VANND_L22_V0342 722.11 BOOL
VANND_L22_V0405 722.09 BOOL
VANND_L22_V0505 722.10 BOOL
VASK_SLANGE 723.12 BOOL  ; SLANGE OENSKES VASKET IC79
VASK_SLANGE_COM_BIT 1150.02 BOOL  ; SLANGE SKAL INNGAA I C79
VENTILFEIL_SIRK_K1 1309.04 BOOL
VENTILFEIL_SIRK_K2 1319.04 BOOL
VENTILFEIL_SIRK_K3 1329.04 BOOL
VS80_K1_HJ_RAP_2STA 901.07 BOOL
VS80_K2_HJ_RAP_2STA 911.07 BOOL
VS80_K3_HJ_RAP_2STA 921.07 BOOL
VST60_K1_KL_INN_N6 2841.08 BOOL
VST60_K1_TR5_N6 2865.02 BOOL
VST60_K2_KL_AVSL 1816.09 BOOL
VST60_K2_KL_INN 1816.08 BOOL
VST80K1_BET_FLOWKONTROLL 1309.07 BOOL  ; BETINGELER START TID FOR FLOWKONTROLL INN
VST80K1_ER_VENT_FLOW D8631 UINT  ; ER- VERDI VENTETID FOER FLOWKONTROLL STARTER
VST80K1_FLOWFEIL 1309.09 BOOL  ; FOR LAV FLOW I RETUR
VST80K1_FLOWKONTROLL 1309.08 BOOL
VST80K1_FLOWKONTROLL_S T0933 BOOL  ; TID MED FOR LAV FLOW I RETUR FOER ALARM SLAAR INN
VST80K1_MAX_DIF_FLOWKONTROLL D8616 UINT  ; MAXIMAL DIFFERANSE MELLOM TUR OG RETURFLOW
VST80K1_PRS_VENT_FLOW D8630 UINT  ; PRS VENTETID FOER FLOWKONTROLL STARTER
VST80K2_BET_FLOWKONTROLL 1319.07 BOOL  ; BETINGELER START TID FOR FLOWKONTROLL INN
VST80K2_ER_VENT_FLOW D8731 UINT  ; ER- VERDI VENTETID FOER FLOWKONTROLL STARTER
VST80K2_FLOWFEIL 1319.09 BOOL  ; FOR LAV FLOW I RETUR
VST80K2_FLOWKONTROLL 1319.08 BOOL
VST80K2_FLOWKONTROLL_S T0934 BOOL  ; TID MED FOR LAV FLOW I RETUR FOER ALARM SLAAR INN
VST80K2_MAX_DIF_FLOWKONTROLL D8716 UINT  ; MAXIMAL DIFFERANSE MELLOM TUR OG RETURFLOW
VST80K2_PRS_VENT_FLOW D8730 UINT  ; PRS VENTETID FOER FLOWKONTROLL STARTER
VST80K3_BET_FLOWKONTROLL 1329.07 BOOL  ; BETINGELER START TID FOR FLOWKONTROLL INN
VST80K3_ER_VENT_FLOW D8801 UINT  ; ER- VERDI VENTETID FOER FLOWKONTROLL STARTER
VST80K3_FLOWFEIL 1329.09 BOOL  ; FOR LAV FLOW I RETUR
VST80K3_FLOWKONTROLL 1329.08 BOOL
VST80K3_FLOWKONTROLL_S T0935 BOOL  ; TID MED FOR LAV FLOW I RETUR FOER ALARM SLAAR INN
VST80K3_MAX_DIF_FLOWKONTROLL D8816 UINT  ; MAXIMAL DIFFERANSE MELLOM TUR OG RETURFLOW
VST80K3_PRS_VENT_FLOW D8800 UINT  ; PRS VENTETID FOER FLOWKONTROLL STARTER
VST80_BIL1_VASKET 701.02 BOOL  ; BENYTTES TIL FLASH PAA VEGG VED BIL 1
VST80_BIL1_VASKET_TID_S T0114 BOOL  ; BENYTTES TIL AA RESET 701.02
VST80_BIL1_VASKET_TID_T 0114 NUMBER  ; BENYTTES TIL AA RESET 701.02
VST80_BIL21_VASKET_TID_S T0116 BOOL  ; BENYTTES TIL AA RESET 705.02
VST80_BIL2_VASKET 705.02 BOOL  ; BENYTTES TIL FLASH PAA VEGG VED BIL 2
VST80_BIL2_VASKET_TID_T 0116 NUMBER  ; BENYTTES TIL AA RESET 705.02
VST80_HENGER1_VASKET 703.02 BOOL  ; BENYTTES TIL FLASH PAA VEGG VED HENGER 1
VST80_HENGER1_VASKET_T 0115 NUMBER  ; BENYTTES TIL AA RESET 703.02
VST80_HENGER1_VASKET_TID_S T0115 BOOL  ; BENYTTES TIL AA RESET 703.02
VST80_HENGER2_VASKET 707.02 BOOL  ; BENYTTES TIL FLASH PAA VEGG VED HENGER 2
VST80_HENGER2_VASKET_T 0117 NUMBER  ; BENYTTES TIL AA RESET 707.02
VST80_HENGER2_VASKET_TID_S T0117 BOOL  ; BENYTTES TIL AA RESET 707.02
VST80_K1R_DIF_S 1308.02 BOOL  ; MENGEDIFFERANSE TUR RETUR FOR STOR
VST80_K1_0_STATUS 500.01 BOOL  ; XX
VST80_K1_0_ST_HJ1 400.00 BOOL
VST80_K1_0_ST_HJ2 400.01 BOOL
VST80_K1_0_ST_HJ3 400.02 BOOL
VST80_K1_1_STATUS 500.02 BOOL  ; Z
VST80_K1_1_ST_HJ1 400.03 BOOL
VST80_K1_1_ST_HJ2 400.04 BOOL  ; Z
VST80_K1_1_ST_HJ3 400.05 BOOL  ; Z
VST80_K1_1_ST_HJ4 400.06 BOOL  ; Z
VST80_K1_1_ST_HJ5 400.07 BOOL  ; Z
VST80_K1_1_ST_HJ6 400.08 BOOL  ; Z
VST80_K1_2_STAT 500.03 BOOL  ; Z
VST80_K1_2_ST_HJ1 400.09 BOOL  ; Z
VST80_K1_2_ST_HJ2 400.10 BOOL  ; Z
VST80_K1_AUT_NOEDSTOPP 1305.04 BOOL  ; NOEDSTOPPSIGNAL FRA VASKESTASJON KURS1
VST80_K1_AVLESE_FLOW D7990 INT
VST80_K1_AVLES_FLOW D8690 INT
VST80_K1_B8011_ER_CT D8040 CHANNEL  ; B8011 -VST80-KURS1. ER-VERDI KONDUKTIVITET I RETUR TIL VST
VST80_K1_B8012_ER_TT D8006 CHANNEL  ; B8012 -VST80-KURS1. ER-VERDI TEMPERATUR I RETUR TIL VST
VST80_K1_B8012_ER_TTR D8604 INT
VST80_K1_B8014_ER_TT D8000 CHANNEL  ; B8014 -VST80-KURS1. ER-VERDI TEMPERATUR I TUR TIL VST
VST80_K1_DIF_HYSTVERDI_OVERSKREDET 1308.01 BOOL  ; BENYTTES TIL AA SKAPE HYSTERESE VED FOR STOR MENDEFORSK. MELLOM TUR OG RETUR  1308.01=0=MENDEDIF OK
VST80_K1_DRIFT 500.00 BOOL  ; XX
VST80_K1_ER_COND D8600 CHANNEL  ; SKAL_RETTES_TIL_K1_KOND_ERVERDI
VST80_K1_FEIL 500.04 BOOL  ; Z
VST80_K1_FEILTID 500.05 BOOL  ; Z
VST80_K1_FORSINK_MENGDEDIF T0151 BOOL  ; TID SOM FORSINKER MENGDEDIF. STOPP AV FASE
VST80_K1_GRM_KONTR_VENT T0884 BOOL  ; VENT MED GRENSEMELKOVERVAAKING
VST80_K1_HJ10 902.01 BOOL
VST80_K1_HJ11 902.02 BOOL
VST80_K1_HJ12 902.03 BOOL
VST80_K1_HJ13 902.04 BOOL
VST80_K1_HJ14 902.05 BOOL
VST80_K1_HJ15 902.06 BOOL
VST80_K1_HJ16 902.07 BOOL
VST80_K1_HJ17 902.08 BOOL
VST80_K1_HJ18 902.09 BOOL
VST80_K1_HJ19 902.10 BOOL
VST80_K1_HJ2 901.09 BOOL
VST80_K1_HJ20 902.11 BOOL
VST80_K1_HJ21 902.12 BOOL
VST80_K1_HJ22 902.13 BOOL
VST80_K1_HJ23 902.15 BOOL
VST80_K1_HJ3 901.10 BOOL
VST80_K1_HJ4 901.11 BOOL
VST80_K1_HJ5 901.12 BOOL
VST80_K1_HJ6 901.13 BOOL
VST80_K1_HJ7 901.14 BOOL
VST80_K1_HJ8 901.15 BOOL
VST80_K1_HJ9 902.00 BOOL
VST80_K1_HYST_D8680 D8682 WORD  ; HYSTERESE VED UTKOBLING AV TURPUMPE PGA. FOR STOR MENGDEFORSKJELL MELLOM TUR OG RETUR I VASKEN
VST80_K1_INDKON 500.06 BOOL  ; Z
VST80_K1_IND_INNE 500.15 BOOL  ; 0=ET INDIVID AKTIVT
VST80_K1_KL_F_REST D4044 CHANNEL  ; START-TIDSPUNKT FOR START AV KLAPRING
VST80_K1_KOELES 300.14 BOOL  ; Z
VST80_K1_KOEPLASS_1 D5000 CHANNEL  ; Z
VST80_K1_KOEPLASS_2 D5002 UDINT  ; Z
VST80_K1_KOEPLASS_3 D5004 UDINT  ; Z
VST80_K1_KOMMANDO_KOE 300.15 BOOL  ; Z
VST80_K1_LINJEFEIL_TXT D4064 CHANNEL
VST80_K1_LUTTID_INN 1309.10 BOOL
VST80_K1_LUT_UTE 1307.09 BOOL  ; LUT UTE AV SYSTEM
VST80_K1_MAX_DIF_TUR_RETUR D8680 WORD  ; MAX DIFERANSE MELLOM TUR OG RETURMENGDE UNDER FORSK.--VASKEM.FASE--HETVANSFASE
VST80_K1_MENGDERESET 1307.04 BOOL  ; RESETTER MENGDETELLER I TUR OG RETUR
VST80_K1_NOEDSTOPP 1305.12 BOOL  ; UTKOBLING AV NIVAA PAA TANK SOM SKAL VASKES
VST80_K1_OFF_IMPULS 500.14 BOOL  ; Z
VST80_K1_ONIMPULS 500.11 BOOL  ; Z
VST80_K1_PAADR D8064 CHANNEL
VST80_K1_PRS_GR_MELK D8620 CHANNEL
VST80_K1_PRS_STERTEMP D8606 CHANNEL
VST80_K1_Q8001_ER_F D8020 CHANNEL  ; Q8001 -VST80-KURS1. ER-VERDI FLOW I TUR
VST80_K1_Q8001_ER_MENDE D8614 WORD  ; '
VST80_K1_Q8001_ER_SIST_MENGDE D8674 WORD  ; MENGDE SISTE ER-VERDI TURSIDE PAA KURSEN
VST80_K1_Q8001_PRS_MENDE D8618 WORD  ; PRS MENGDE SOM STYRER P8001 VED FASESKIFTE
VST80_K1_Q8001_PRS_TIL_TANK D8676 UINT  ; MENGDE  PRS  MENDE FRAM TIL TANK
VST80_K1_Q8001_PRS_TR2 D8678 WORD  ; PRESET TIL TANK TR2
VST80_K1_Q8017_ER_MENGDE D8626 WORD  ; MENGDE I RETUR PAA  KURS  ER_VERDI
VST80_K1_RA_FLOW D8690 CHANNEL  ; -VST80-KURS1. VASKERAPPORT.  FLOW
VST80_K1_RESET 500.09 BOOL  ; Z
VST80_K1_R_Q8011_ER_F D8030 CHANNEL  ; Q8011 -VST80-KURS1 . ER-VERDI FLOW I RETUR
VST80_K1_SPERR_HR H1.01 BOOL  ; RETENTETIV FUNKSJON
VST80_K1_START 500.07 BOOL  ; Z
VST80_K1_STARTIMPULS 500.10 BOOL  ; Z
VST80_K1_STATUS D7640 CHANNEL  ; OPPSAMLING AV VASKESTATUS UNDER VASK
VST80_K1_SYRE_FRAM_BOERVERDI D8646 DWORD  ; SYRE TIL VASKEKULE. BOER VERDI VED START. VERDI FRA D8644
VST80_K1_SYRE_FRAM_TR18 C0150 BOOL  ; FRAMKJOERING AV SYRE FRAM TIL VASKEKULE FOER SYREFASE
VST80_K1_SYRE_VED_TANK 1308.04 BOOL  ; SYRE UTE VED VASKEKULE ETTER SKYLLEFASE
VST80_K1_T82_LAVCOND 1308.11 BOOL  ; KURS1  FASE LUT INN KONSENTRASJON T82 FOR LAV
VST80_K1_T84_LAVCOND 1308.12 BOOL  ; KURS1  FASE LUT INN KONSENTRASJON T84 FOR LAV
VST80_K1_TEKST_BILDE D8692 CHANNEL
VST80_K1_TID_LUT_UTE T0881 BOOL  ; VENTETID FOER LUT UTE AV SYSTEM REGISTRERES
VST80_K1_TID_S T0500 BOOL  ; Z
VST80_K1_TID_T 0500 NUMBER  ; Z
VST80_K1_TID_TR1 D4001 CHANNEL
VST80_K1_TID_TR10 D4010 CHANNEL
VST80_K1_TID_TR11 D4011 CHANNEL
VST80_K1_TID_TR12 D4012 CHANNEL
VST80_K1_TID_TR13 D4013 CHANNEL
VST80_K1_TID_TR14 D4014 CHANNEL
VST80_K1_TID_TR15 D4015 CHANNEL
VST80_K1_TID_TR16 D4016 CHANNEL
VST80_K1_TID_TR17 D4017 CHANNEL
VST80_K1_TID_TR18 D4018 CHANNEL
VST80_K1_TID_TR19 D4019 CHANNEL
VST80_K1_TID_TR2 D4002 CHANNEL
VST80_K1_TID_TR20 D4020 CHANNEL
VST80_K1_TID_TR21 D4021 CHANNEL
VST80_K1_TID_TR22 D4022 CHANNEL
VST80_K1_TID_TR23 D4023 CHANNEL
VST80_K1_TID_TR24 D4024 CHANNEL
VST80_K1_TID_TR25 D4025 CHANNEL
VST80_K1_TID_TR26 D4026 CHANNEL
VST80_K1_TID_TR27 D4027 CHANNEL
VST80_K1_TID_TR28 D4028 CHANNEL
VST80_K1_TID_TR29 D4029 CHANNEL
VST80_K1_TID_TR3 D4003 CHANNEL
VST80_K1_TID_TR30 D4030 CHANNEL
VST80_K1_TID_TR4 D4004 CHANNEL
VST80_K1_TID_TR5 D4005 CHANNEL
VST80_K1_TID_TR6 D4006 CHANNEL
VST80_K1_TID_TR7 D4007 CHANNEL
VST80_K1_TID_TR8 D4008 CHANNEL
VST80_K1_TID_TR9 D4009 CHANNEL
VST80_K1_TIL_TANK_OK 1308.09 BOOL
VST80_K1_TMU 500.08 BOOL  ; Z
VST80_K1_TMU_TID_S T0700 BOOL  ; MAX-TID TMU OM IKKE LINJE LEGGES
VST80_K1_TMU_TID_T 0700 NUMBER  ; MAX-TID TMU OM IKKE LINJE LEGGES
VST80_K1_TRINN_HJ1 D4062 CHANNEL
VST80_K1_TRINN_NR D4060 CHANNEL  ; ANGIR VASKETRINN SOM VASKEN ER I
VST80_K1_UPROG_1 1301.00 BOOL
VST80_K1_UPROG_2 1301.01 BOOL
VST80_K1_UPROG_3 1301.02 BOOL
VST80_K1_UPROG_4 1301.03 BOOL
VST80_K1_UPROG_5 1301.04 BOOL
VST80_K1_UPROG_6 1301.05 BOOL
VST80_K1_V8211_SLUK_LUTUTSKYLL 1308.05 BOOL  ; V8211  TIL SLUK I LUT-SKYLL ETTER AT  KONSENTRASJONEN HAR VAERT UNDER  GRENSEVERDI
VST80_K1_V8311_SLUK_SYREUTSKYLL 1308.06 BOOL  ; V8311  TIL SLUK ISYRE-SKYLL ETTER AT  KONSENTRASJONEN HAR VAERT UNDER  GRENSEVERDI
VST80_K1_VALGT 1307.11 BOOL
VST80_K1_VALGT_IMP 1307.12 BOOL
VST80_K1_VRAP_RESET T0120 BOOL  ; RESETTER INFO I VASKERAPPORT FOR KURS1
VST80_K2R_DIF_S 1318.02 BOOL  ; MENGEDIFFERANSE TUR RETUR FOR STOR
VST80_K2_0_STATUS 501.01 BOOL  ; XX
VST80_K2_0_STAT_HJ0 401.04 BOOL  ; Z
VST80_K2_1_STATUS 501.02 BOOL  ; Z
VST80_K2_1_STAT_HJ0 401.05 BOOL
VST80_K2_2_STAT 501.03 BOOL  ; Z
VST80_K2_2_STAT_HJ0 401.06 BOOL
VST80_K2_AUT_NOEDSTOPP 1315.04 BOOL  ; NOEDSTOPPSIGNAL FRA VASKESTASJON KURS2
VST80_K2_AVLESE_FLOW D7992 INT
VST80_K2_B8021_ER_CT D8042 CHANNEL  ; B8021 -VST80-KURS2. ER-VERDI KONDUKTIVITET I RETUR TIL VST
VST80_K2_B8022_ER_TT D8008 CHANNEL  ; B8022 -VST80-KURS2. ER-VERDI TEMPERATUR I RETUR TIL VST
VST80_K2_B8024_ER_TT D8002 CHANNEL  ; B8024 -VST80-KURS2. ER-VERDI TEMPERATUR I TUR TIL VST
VST80_K2_C_0_ST_HJ1 932.05 BOOL
VST80_K2_C_0_ST_HJ2 932.06 BOOL
VST80_K2_C_0_ST_HJ3 932.07 BOOL
VST80_K2_C_1_ST_HJ1 932.08 BOOL
VST80_K2_C_1_ST_HJ2 932.09 BOOL
VST80_K2_C_1_ST_HJ3 932.10 BOOL
VST80_K2_C_1_ST_HJ4 932.11 BOOL
VST80_K2_C_1_ST_HJ5 932.12 BOOL
VST80_K2_C_1_ST_HJ6 932.13 BOOL
VST80_K2_C_2_ST_HJ1 932.14 BOOL
VST80_K2_C_BIL_0_ST_HJ1 932.02 BOOL
VST80_K2_C_BIL_0_ST_HJ2 932.03 BOOL
VST80_K2_DRIFT 501.00 BOOL  ; XX
VST80_K2_FEILTID 501.05 BOOL  ; Z
VST80_K2_FORSINK_MENGDEDIF T0251 BOOL
VST80_K2_GRM_KONTR_VENT T0894 BOOL  ; VENT MED GRENSEMELKOVERVAAKING
VST80_K2_GR_IND_HJ1 401.10 BOOL  ; INVERTERT INDIVIDADRESSE FOR EN GRUPPE INDIVIDER
VST80_K2_GR_IND_HJ2 401.11 BOOL  ; INVERTERT INDIVIDADRESSE FOR EN GRUPPE INDIVIDER
VST80_K2_GR_IND_HJ3 401.12 BOOL  ; INVERTERT INDIVIDADRESSE FOR EN GRUPPE INDIVIDER
VST80_K2_HJ10 912.01 BOOL
VST80_K2_HJ11 912.02 BOOL
VST80_K2_HJ12 912.03 BOOL
VST80_K2_HJ13 912.04 BOOL
VST80_K2_HJ16 912.07 BOOL
VST80_K2_HJ17 912.08 BOOL
VST80_K2_HJ2 911.09 BOOL
VST80_K2_HJ21 912.12 BOOL
VST80_K2_HJ22 912.13 BOOL
VST80_K2_HJ23 912.15 BOOL
VST80_K2_HJ3 911.10 BOOL
VST80_K2_HJ4 911.11 BOOL
VST80_K2_HJ5 911.12 BOOL
VST80_K2_HJ6 911.13 BOOL
VST80_K2_HJ7 911.14 BOOL
VST80_K2_HJ8 911.15 BOOL  ; 92115
VST80_K2_HJ9 912.00 BOOL
VST80_K2_INDKON 501.06 BOOL  ; Z
VST80_K2_IND_INNE 501.15 BOOL  ; Z
VST80_K2_IND_INNE_HJ1 401.00 BOOL
VST80_K2_IND_INNE_HJ2 401.01 BOOL
VST80_K2_IND_INNE_HJ3 401.02 BOOL
VST80_K2_KL_F_REST D4144 CHANNEL  ; START-TIDSPUNKT FOR START AV KLAPRING
VST80_K2_KOEPLASS_1 D5010 CHANNEL  ; PGM501_KOEPLASS_1
VST80_K2_KOEPLASS_2 D5012 UDINT  ; PGM501_KOEPLASS_2
VST80_K2_KOEPLASS_3 D5014 UDINT  ; PGM501_KOEPLASS_3
VST80_K2_LINJEFEIL_TXT D4164 CHANNEL
VST80_K2_LUTTID_INN 1319.10 BOOL
VST80_K2_LUT_UTE 1317.09 BOOL
VST80_K2_MENGDERESET 1317.04 BOOL  ; RESETTER MENGDETELLER I TUR OG RETUR
VST80_K2_NOEDSTOPP 1315.12 BOOL  ; UTKOBLING AV NIVAA PAA TANK SOM SKAL VASKES
VST80_K2_OFF_IMPULS 501.14 BOOL  ; Z
VST80_K2_ONIMPULS 501.11 BOOL  ; Z
VST80_K2_PAADR D8164 CHANNEL
VST80_K2_PRS_GR_MELK D8720 INT
VST80_K2_PRS_STERTEMP D8706 CHANNEL
VST80_K2_Q8002_ER_F D8022 CHANNEL  ; Q8002 -VST80-KURS2. ER-VERDI FLOW I TUR
VST80_K2_Q8002_ER_MENDE D8714 INT
VST80_K2_Q8002_ER_SIST_MENGDE D8774 CHANNEL
VST80_K2_Q8002_PRS_MENDE D8718 WORD  ; PRS MENGDE SOM STYRER P8002VED FASESKIFTE
VST80_K2_Q8002_PRS_TIL_TANK D8776 INT
VST80_K2_Q8002_PRS_TR2 D8778 INT
VST80_K2_RA_FLOW D8790 CHANNEL  ; -VST80-KURS2 . VASKERAPPORT.  FLOW
VST80_K2_RESET 501.09 BOOL  ; Z
VST80_K2_R_Q8012_ER_F D8032 CHANNEL  ; Q8012 -VST80-KURS2. ER-VERDI FLOW I RETUR
VST80_K2_SIRKULASJON_ 1319.00 BOOL
VST80_K2_SPERR_HR H1.02 BOOL  ; RETENTETIV FUNKSJON
VST80_K2_START 501.07 BOOL  ; Z
VST80_K2_STARTIMPULS 501.10 BOOL  ; Z
VST80_K2_STARTKOMMANDO 401.14 BOOL  ; Z
VST80_K2_START_FRA_N1 401.13 BOOL  ; STARTSIGNAL FRA NODE1 FOR C06-C07-C08-C50-C52-C53
VST80_K2_STATUS D7740 CHANNEL  ; OPPSAMLING AV VASKESTATUS UNDER VASK
VST80_K2_SYRE_FRAM_TR18 C0250 BOOL  ; FRAMKJOERING AV SYRE FRAM TIL VASKEKULE FOER SYREFASE
VST80_K2_SYRE_VED_TANK 1318.04 BOOL  ; SYRE UTE VED VASKEKULE ETTER SKYLLEFASE
VST80_K2_T82_LAVCOND 1318.11 BOOL  ; KURS2  FASE LUT INN KONSENTRASJON T82 FOR LAV
VST80_K2_T84_LAVCOND 1318.12 BOOL  ; KURS2  FASE LUT INN KONSENTRASJON T84 FOR LAV
VST80_K2_TEKST_BILDE D8792 CHANNEL
VST80_K2_TID_LUT_UTE T0882 BOOL  ; VENTETID FOER LUT UTE AV SYSTEM REGISTRERES
VST80_K2_TID_S T0501 BOOL  ; Z
VST80_K2_TID_T 0501 NUMBER  ; Z
VST80_K2_TID_TR1 D4101 CHANNEL
VST80_K2_TID_TR10 D4110 CHANNEL
VST80_K2_TID_TR11 D4111 CHANNEL
VST80_K2_TID_TR12 D4112 CHANNEL
VST80_K2_TID_TR13 D4113 CHANNEL
VST80_K2_TID_TR14 D4114 CHANNEL
VST80_K2_TID_TR15 D4115 CHANNEL
VST80_K2_TID_TR16 D4116 CHANNEL
VST80_K2_TID_TR17 D4117 CHANNEL
VST80_K2_TID_TR18 D4118 CHANNEL
VST80_K2_TID_TR19 D4119 CHANNEL
VST80_K2_TID_TR2 D4102 CHANNEL
VST80_K2_TID_TR20 D4120 CHANNEL
VST80_K2_TID_TR21 D4121 CHANNEL
VST80_K2_TID_TR22 D4122 CHANNEL
VST80_K2_TID_TR23 D4123 CHANNEL
VST80_K2_TID_TR24 D4124 CHANNEL
VST80_K2_TID_TR25 D4125 CHANNEL
VST80_K2_TID_TR26 D4126 CHANNEL
VST80_K2_TID_TR27 D4127 CHANNEL
VST80_K2_TID_TR28 D4128 CHANNEL
VST80_K2_TID_TR29 D4129 CHANNEL
VST80_K2_TID_TR3 D4103 CHANNEL
VST80_K2_TID_TR30 D4130 CHANNEL
VST80_K2_TID_TR4 D4104 CHANNEL
VST80_K2_TID_TR5 D4105 CHANNEL
VST80_K2_TID_TR6 D4106 CHANNEL
VST80_K2_TID_TR7 D4107 CHANNEL
VST80_K2_TID_TR8 D4108 CHANNEL
VST80_K2_TID_TR9 D4109 CHANNEL
VST80_K2_TIL_TANK_OK 1318.09 BOOL
VST80_K2_TMU 501.08 BOOL
VST80_K2_TMU_TID_S T0701 BOOL  ; MAX-TID TMU OM IKKE LINJE LEGGES
VST80_K2_TMU_TID_T 0701 NUMBER  ; MAX-TID TMU OM IKKE LINJE LEGGES
VST80_K2_TRINN_HJ1 D4162 CHANNEL
VST80_K2_TRINN_NR D4160 CHANNEL  ; ANGIR VASKETRINN SOM VASKEN ER I
VST80_K2_UPROG_1 1311.00 BOOL
VST80_K2_UPROG_10 1311.09 BOOL
VST80_K2_UPROG_11 1311.10 BOOL
VST80_K2_UPROG_2 1311.01 BOOL
VST80_K2_UPROG_3 1311.02 BOOL
VST80_K2_UPROG_4 1311.03 BOOL
VST80_K2_UPROG_5 1311.04 BOOL
VST80_K2_UPROG_6 1311.05 BOOL
VST80_K2_UPROG_7 1311.06 BOOL
VST80_K2_UPROG_8 1311.07 BOOL
VST80_K2_UPROG_9 1311.08 BOOL
VST80_K2_V8212_SLUK_LUTUTSKYLL 1318.15 BOOL  ; V8212  TIL SLUK I LUT-SKYLL ETTER AT  KONSENTRASJONEN HAR VAERT UNDER  GRENSEVERDI
VST80_K2_V8412_SLUK_SYREUTSKYLL 1318.06 BOOL  ; V8412  TIL SLUK ISYRE-SKYLL ETTER AT  KONSENTRASJONEN HAR VAERT UNDER  GRENSEVERDI
VST80_K2_VALGT 1317.11 BOOL
VST80_K2_VALGT_IMP 1317.12 BOOL
VST80_K2_VRAP_RESET T0130 BOOL
VST80_K3R_DIF_S 1328.02 BOOL
VST80_K3_0_STATUS 502.01 BOOL  ; XX
VST80_K3_0_STAT_HJ0 402.04 BOOL  ; Z
VST80_K3_1_STATUS 502.02 BOOL  ; Z
VST80_K3_1_STAT_HJ0 402.05 BOOL  ; Z
VST80_K3_AUT_NOEDSTOPP 1325.04 BOOL  ; NOEDSTOPPSIGNAL FRA VASKESTASJON KURS3
VST80_K3_AVLESE_FLOW D7994 INT
VST80_K3_B8031_ER_CT D8044 CHANNEL  ; B8031 -VST80-KURS3. ER-VERDI KONDUKTIVITET I RETUR TIL VST
VST80_K3_B8032_ER_TT D8010 CHANNEL  ; B8032 -VST80-KURS3. ER-VERDI TEMPERATUR I RETUR TIL VST
VST80_K3_B8034_ER_TT D8004 CHANNEL  ; B8034 -VST80-KURS3. ER-VERDI TEMPERATUR I TUR TIL VST
VST80_K3_DRIFT 502.00 BOOL  ; XX
VST80_K3_FEILTID 502.05 BOOL  ; Z
VST80_K3_FORSINK_MENGDEDIF T0351 BOOL
VST80_K3_GRM_KONTR_VENT T0904 BOOL  ; VENT MED GRENSEMELKOVERVAAKING
VST80_K3_HJ10 922.01 BOOL
VST80_K3_HJ11 922.02 BOOL
VST80_K3_HJ12 922.03 BOOL
VST80_K3_HJ13 922.04 BOOL
VST80_K3_HJ16 922.07 BOOL
VST80_K3_HJ17 922.08 BOOL
VST80_K3_HJ2 921.09 BOOL
VST80_K3_HJ21 922.12 BOOL
VST80_K3_HJ22 922.13 BOOL
VST80_K3_HJ3 921.10 BOOL
VST80_K3_HJ4 921.11 BOOL
VST80_K3_HJ5 921.12 BOOL
VST80_K3_HJ6 921.13 BOOL
VST80_K3_HJ7 921.14 BOOL
VST80_K3_HJ8 921.15 BOOL
VST80_K3_HJ9 922.00 BOOL
VST80_K3_INDKON 502.06 BOOL  ; Z
VST80_K3_IND_INNE 502.15 BOOL  ; Z
VST80_K3_IND_INNE_HJ1 402.00 BOOL
VST80_K3_IND_INNE_HJ2 402.01 BOOL
VST80_K3_IND_INNE_HJ3 402.02 BOOL
VST80_K3_KLAPRING 1326.08 BOOL
VST80_K3_KLAP_SLUTT 1326.09 BOOL  ; KLAPRING I FASEN AVSLUTTET.
VST80_K3_KL_F_REST D4244 CHANNEL  ; START-TIDSPUNKT FOR START AV KLAPRING
VST80_K3_KOEPLASS_1 D5020 CHANNEL  ; PGM 502 KOEPLASS 1
VST80_K3_KOEPLASS_2 D5022 UDINT  ; PGM 502 KOEPLASS 2
VST80_K3_KOEPLASS_3 D5024 UDINT  ; PGM502_KOEPLASS_3
VST80_K3_LINJEFEIL_TXT D4264 CHANNEL
VST80_K3_LUTTID_INN 1329.10 BOOL
VST80_K3_LUT_UTE 1327.09 BOOL
VST80_K3_MENGDERESET 1327.04 BOOL  ; RESETTER MENGDETELLER I TUR OG RETUR
VST80_K3_NOEDSTOPP 1325.12 BOOL  ; UTKOBLING AV NIVAA PAA TANK SOM SKAL VASKES
VST80_K3_OFF_IMPULS 502.14 BOOL  ; Z
VST80_K3_ONIMPULS 502.11 BOOL  ; Z
VST80_K3_PAADR D8264 CHANNEL
VST80_K3_PRS_GR_MELK D8820 INT
VST80_K3_PRS_STERTEMP D8806 UINT
VST80_K3_Q8003_ER_F D8024 CHANNEL  ; Q8003 -VST80-KURS3. ER-VERDI FLOW I TUR
VST80_K3_Q8003_ER_MENDE D8814 INT
VST80_K3_Q8003_ER_SIST_MENGDE D8874 CHANNEL
VST80_K3_Q8003_PRS_MENDE D8818 WORD  ; PRS MENGDE SOM STYRER P8003 VED FASESKIFTE
VST80_K3_Q8003_PRS_TIL_TANK D8876 CHANNEL
VST80_K3_Q8003_PRS_TR2 D8878 INT
VST80_K3_Q8013_ER_F D8034 CHANNEL  ; Q8013 -VST80-KURS3. ER-VERDI FLOW I RETUR
VST80_K3_RA_FLOW D8890 CHANNEL  ; -VST80-KURS3 . VASKERAPPORT.  FLOW
VST80_K3_RESET 502.09 BOOL  ; PGM502_STOPP
VST80_K3_SILOKL_INN 1328.13 BOOL net:
$?St$Bk?_#[6]
kLAPRING AV 4" LEDNING UNDER SILOVASK INNKOBLET$?St$Bk?_#[6];
VST80_K3_SILO_TOM  ; TEST

## Program NewProgram1 (cyclic task 0)
Local symbols
B0104_TT_ISVRETUR_INT INT
B2114_PT D3120 INT
B2114_PT_FLT1 D10120 REAL
D REAL
DD3010 UDINT
L UINT
NODE28_TELLER CHANNEL
P2101_PÅDRAG_P2101_PRS_FRYS CHANNEL
P2102_PÅDRAG CHANNEL
P2104_PÅDRAG_real REAL
P2201_PRS_FRYS CHANNEL
P23_ISV_DIFF_TRYKK UINT
PGM504_IND_C23 BOOL
PGM554_2_STATUS BOOL
SEP21_FRYSER BOOL
VST80_K3_AVLES_FLOW CHANNEL
VST80_K8_AVLES_FLOW CHANNEL
cfd113 BOOL
cxf113 BOOL
dummy BOOL
f113 BOOL
f135010 BOOL
p2060_ut BOOL
p2101_P UINT
p2101_pådrag_P2101_PRS_FRYS CHANNEL

### Section PROFIBUSKOMMUNIKASJON

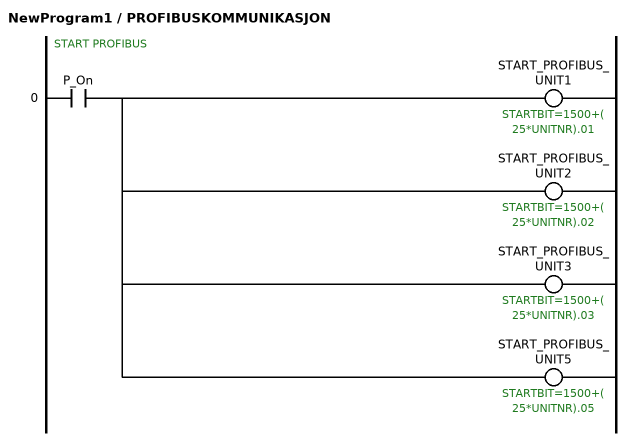
; rung 0: START PROFIBUS
LD P_On
OUT START_PROFIBUS_UNIT1  ; STARTBIT=1500+(25*UNITNR).01
OUT START_PROFIBUS_UNIT2  ; STARTBIT=1500+(25*UNITNR).02
OUT START_PROFIBUS_UNIT3  ; STARTBIT=1500+(25*UNITNR).03
OUT START_PROFIBUS_UNIT5  ; STARTBIT=1500+(25*UNITNR).05

### Section PROFIBUS_N5

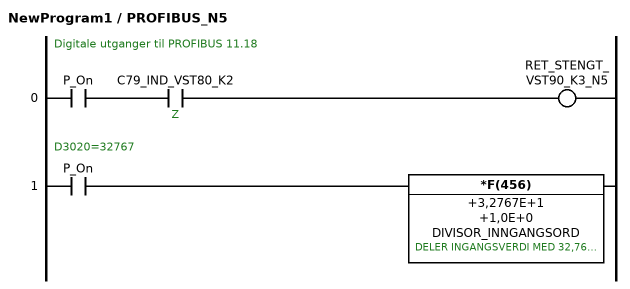
; rung 0: Digitale utganger til PROFIBUS 11.18
LD P_On
AND C79_IND_VST80_K2  ; Z
OUT RET_STENGT_VST90_K3_N5
; rung 1: D3020=32767
LD P_On
*F(456) +3,2767E+1 +1,0E+0 DIVISOR_INNGANGSORD  ; DELER INGANGSVERDI MED 32,760 FOR OMREGNING TIL 0-1000

### Section SEND_FRA_N4

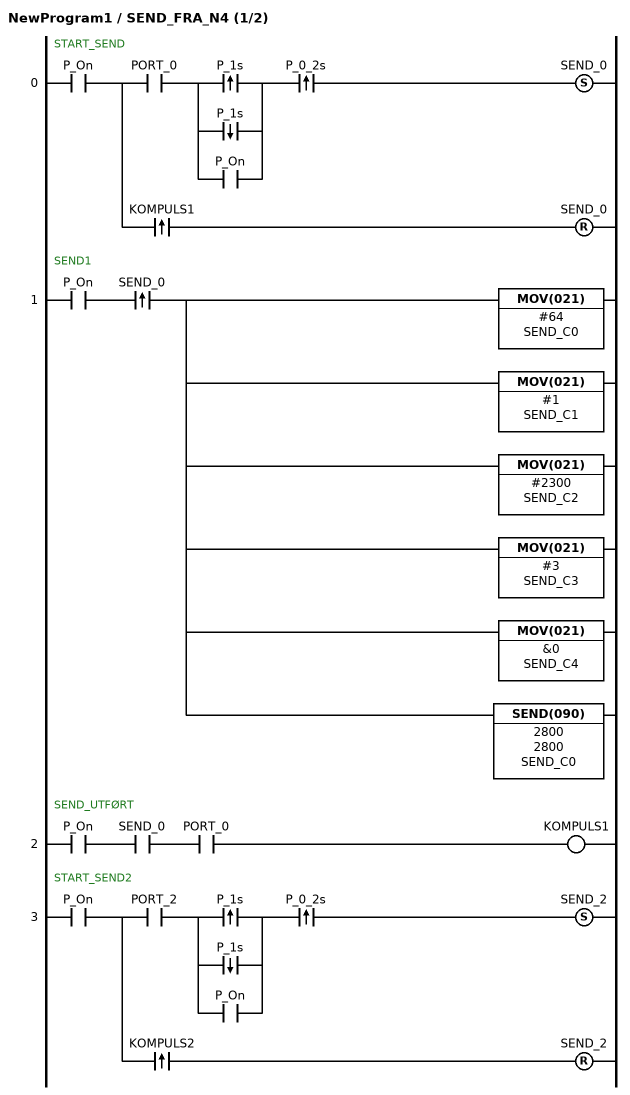
; rung 0: START_SEND
LD P_On
OUT TR0
AND PORT_0
@LD P_1s
%OR P_1s
OR P_On
ANDLD
@AND P_0_2s
SET SEND_0
LD TR0
@AND KOMPULS1
RSET SEND_0
; rung 1: SEND1
LD P_On
@AND SEND_0
MOV(021) #64 SEND_C0
MOV(021) #1 SEND_C1
MOV(021) #2300 SEND_C2
MOV(021) #3 SEND_C3
MOV(021) &0 SEND_C4
SEND(090) 2800 2800 SEND_C0
; rung 2: SEND_UTFØRT
LD P_On
AND SEND_0
AND PORT_0
OUT KOMPULS1
; rung 3: START_SEND2
LD P_On
OUT TR0
AND PORT_2
@LD P_1s
%OR P_1s
OR P_On
ANDLD
@AND P_0_2s
SET SEND_2
LD TR0
@AND KOMPULS2
RSET SEND_2

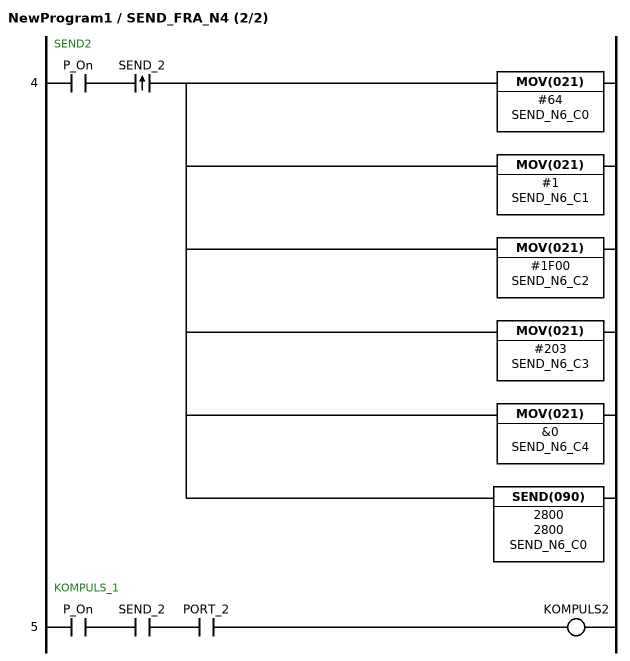
; rung 4: SEND2
LD P_On
@AND SEND_2
MOV(021) #64 SEND_N6_C0
MOV(021) #1 SEND_N6_C1
MOV(021) #1F00 SEND_N6_C2
MOV(021) #203 SEND_N6_C3
MOV(021) &0 SEND_N6_C4
SEND(090) 2800 2800 SEND_N6_C0
; rung 5: KOMPULS_1
LD P_On
AND SEND_2
AND PORT_2
OUT KOMPULS2

### Section KOMMANDO_FEILRESET

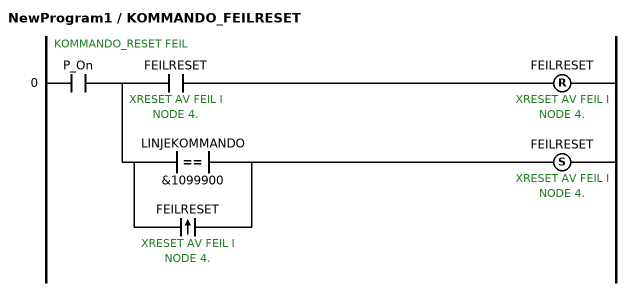
; rung 0: KOMMANDO_RESET FEIL
LD P_On
OUT TR0
AND FEILRESET  ; XRESET AV FEIL I NODE 4.
RSET FEILRESET  ; XRESET AV FEIL I NODE 4.
LD TR0
LD=L(301) LINJEKOMMANDO &1099900
@OR FEILRESET  ; XRESET AV FEIL I NODE 4.
ANDLD
SET FEILRESET  ; XRESET AV FEIL I NODE 4.

### Section K0MMANO
; UTG: 10-03-97 / OVERFØRER KOMMANDOORD FRA INTOUCH TIL PLS-SYSTEM / INTOUC-ADRESSE LINJEVALG: DM3004 / PLS-ADRESSE LINJEVALG:       DM3000 / INTOUCHADRESSE-OBJEKT:     DM3006 / PLS-ADRESSE OBJEKTVALG:    DM3002

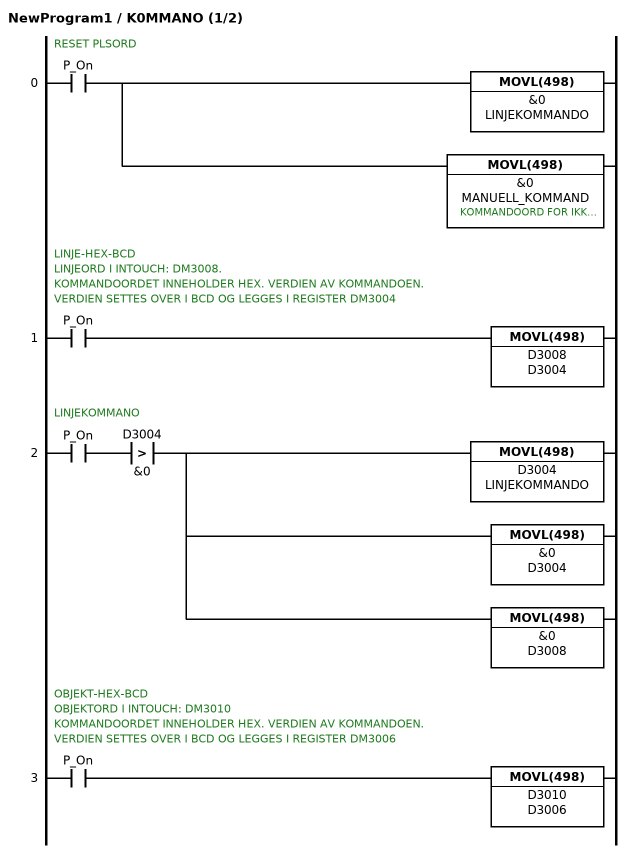
; rung 0: RESET PLSORD
LD P_On
MOVL(498) &0 LINJEKOMMANDO
MOVL(498) &0 MANUELL_KOMMAND  ; KOMMANDOORD FOR IKKE LINJEKOMMANDOER
; rung 1: LINJE-HEX-BCD / LINJEORD I INTOUCH: DM3008. / KOMMANDOORDET INNEHOLDER HEX. VERDIEN AV KOMMANDOEN. / VERDIEN SETTES OVER I BCD OG LEGGES I REGISTER DM3004
LD P_On
MOVL(498) D3008 D3004
; rung 2: LINJEKOMMANO
LD P_On
AND>(320) D3004 &0
MOVL(498) D3004 LINJEKOMMANDO
MOVL(498) &0 D3004
MOVL(498) &0 D3008
; rung 3: OBJEKT-HEX-BCD / OBJEKTORD I INTOUCH: DM3010 / KOMMANDOORDET INNEHOLDER HEX. VERDIEN AV KOMMANDOEN. / VERDIEN SETTES OVER I BCD OG LEGGES I REGISTER DM3006
LD P_On
MOVL(498) D3010 D3006

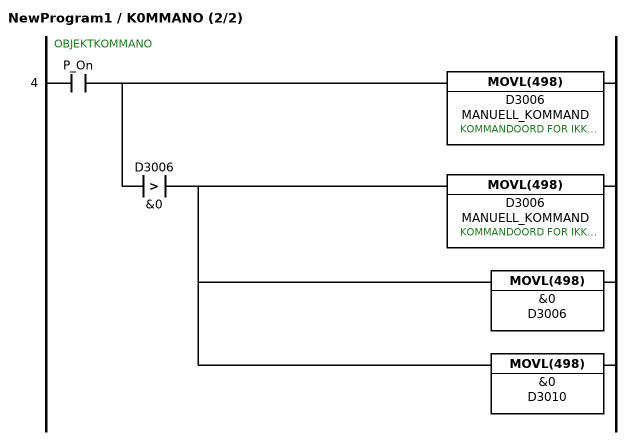
; rung 4: OBJEKTKOMMANO
LD P_On
MOVL(498) D3006 MANUELL_KOMMAND  ; KOMMANDOORD FOR IKKE LINJEKOMMANDOER
AND>(320) D3006 &0
MOVL(498) D3006 MANUELL_KOMMAND  ; KOMMANDOORD FOR IKKE LINJEKOMMANDOER
MOVL(498) &0 D3006
MOVL(498) &0 D3010

### Section N4_X_KOBL_MELLOM_NODER

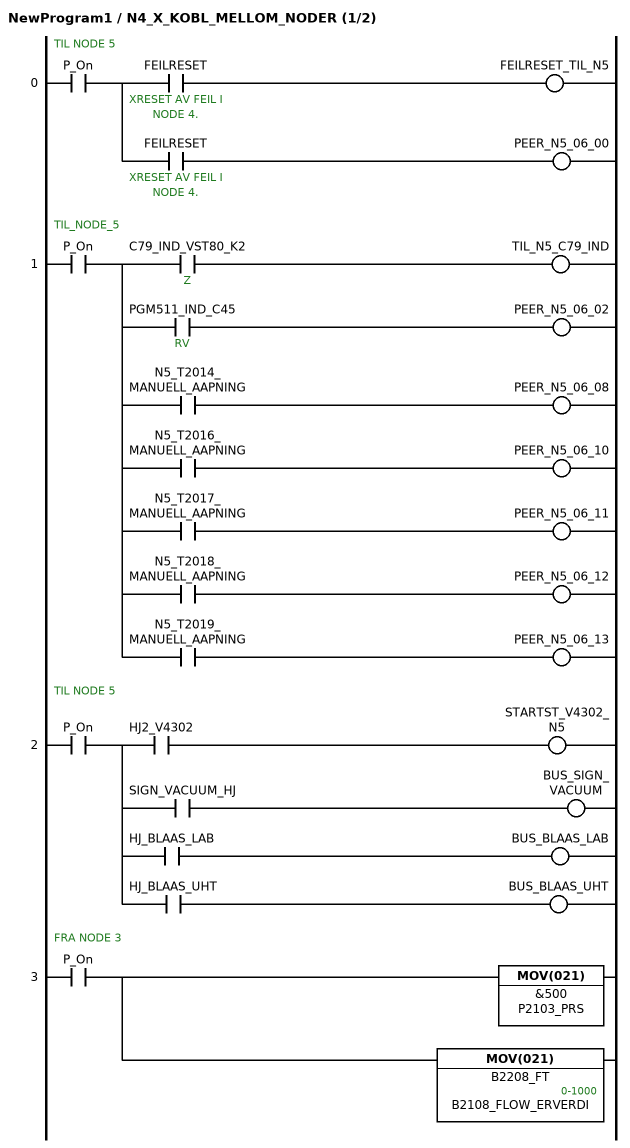
; rung 0: TIL NODE 5
LD P_On
OUT TR0
AND FEILRESET  ; XRESET AV FEIL I NODE 4.
OUT FEILRESET_TIL_N5
LD TR0
AND FEILRESET  ; XRESET AV FEIL I NODE 4.
OUT PEER_N5_06_00
; rung 1: TIL_NODE_5
LD P_On
OUT TR0
AND C79_IND_VST80_K2  ; Z
OUT TIL_N5_C79_IND
LD TR0
AND PGM511_IND_C45  ; RV
OUT PEER_N5_06_02
LD TR0
AND N5_T2014_MANUELL_AAPNING
OUT PEER_N5_06_08
LD TR0
AND N5_T2016_MANUELL_AAPNING
OUT PEER_N5_06_10
LD TR0
AND N5_T2017_MANUELL_AAPNING
OUT PEER_N5_06_11
LD TR0
AND N5_T2018_MANUELL_AAPNING
OUT PEER_N5_06_12
LD TR0
AND N5_T2019_MANUELL_AAPNING
OUT PEER_N5_06_13
; rung 2: TIL NODE 5
LD P_On
OUT TR0
AND HJ2_V4302
OUT STARTST_V4302_N5
LD TR0
AND SIGN_VACUUM_HJ
OUT BUS_SIGN_VACUUM
LD TR0
AND HJ_BLAAS_LAB
OUT BUS_BLAAS_LAB
LD TR0
AND HJ_BLAAS_UHT
OUT BUS_BLAAS_UHT
; rung 3: FRA NODE 3
LD P_On
MOV(021) &500 P2103_PRS
MOV(021) B2208_FT B2108_FLOW_ERVERDI  ; 0-1000

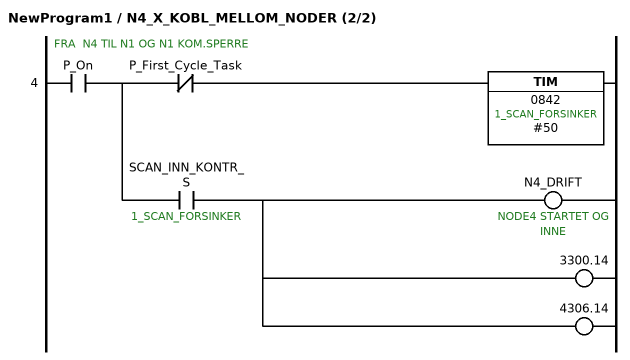
; rung 4: FRA  N4 TIL N1 OG N1 KOM.SPERRE
LD P_On
OUT TR0
ANDNOT P_First_Cycle_Task
TIM 0842 #50  ; 1_SCAN_FORSINKER
LD TR0
AND SCAN_INN_KONTR_S  ; 1_SCAN_FORSINKER
OUT N4_DRIFT  ; NODE4 STARTET OG INNE
OUT 3300.14
OUT 4306.14

### Section INTERNBRUK_GRAFIKK

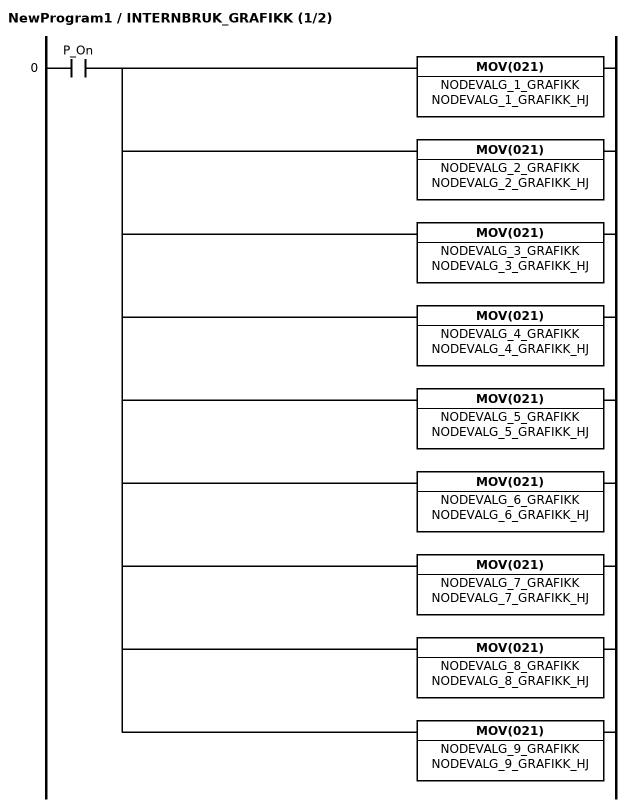
; rung 0
LD P_On
MOV(021) NODEVALG_1_GRAFIKK NODEVALG_1_GRAFIKK_HJ
MOV(021) NODEVALG_2_GRAFIKK NODEVALG_2_GRAFIKK_HJ
MOV(021) NODEVALG_3_GRAFIKK NODEVALG_3_GRAFIKK_HJ
MOV(021) NODEVALG_4_GRAFIKK NODEVALG_4_GRAFIKK_HJ
MOV(021) NODEVALG_5_GRAFIKK NODEVALG_5_GRAFIKK_HJ
MOV(021) NODEVALG_6_GRAFIKK NODEVALG_6_GRAFIKK_HJ
MOV(021) NODEVALG_7_GRAFIKK NODEVALG_7_GRAFIKK_HJ
MOV(021) NODEVALG_8_GRAFIKK NODEVALG_8_GRAFIKK_HJ
MOV(021) NODEVALG_9_GRAFIKK NODEVALG_9_GRAFIKK_HJ

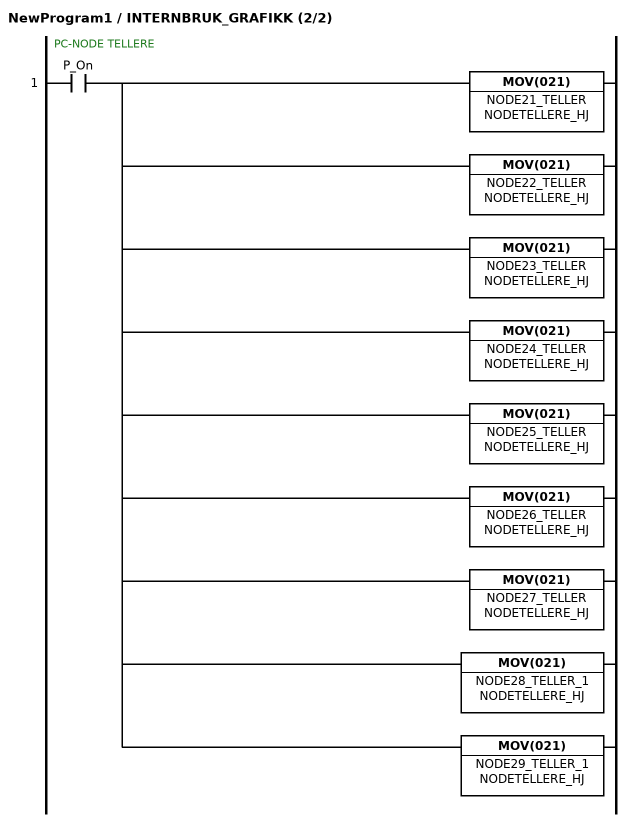
; rung 1: PC-NODE TELLERE
LD P_On
MOV(021) NODE21_TELLER NODETELLERE_HJ
MOV(021) NODE22_TELLER NODETELLERE_HJ
MOV(021) NODE23_TELLER NODETELLERE_HJ
MOV(021) NODE24_TELLER NODETELLERE_HJ
MOV(021) NODE25_TELLER NODETELLERE_HJ
MOV(021) NODE26_TELLER NODETELLERE_HJ
MOV(021) NODE27_TELLER NODETELLERE_HJ
MOV(021) NODE28_TELLER_1 NODETELLERE_HJ
MOV(021) NODE29_TELLER_1 NODETELLERE_HJ

### Section PLS_STARTIND_OG_BLINK

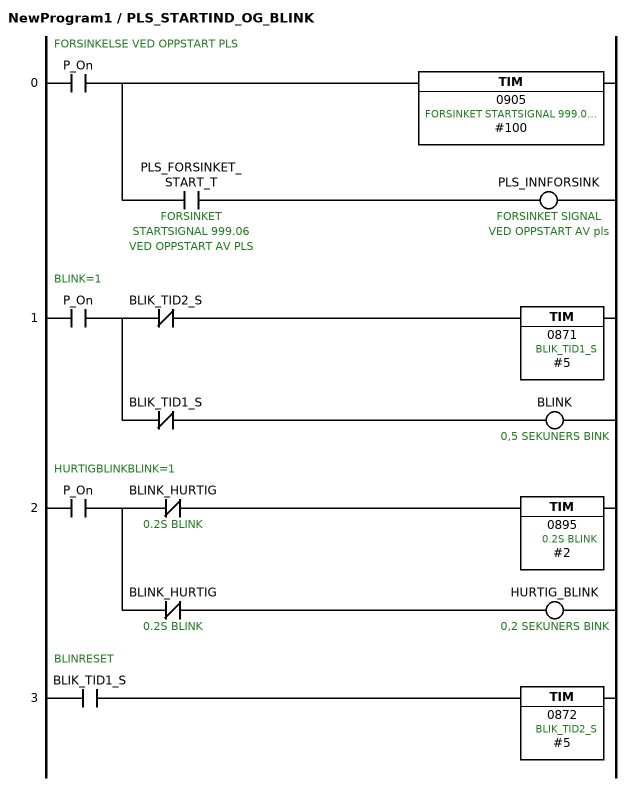
; rung 0: FORSINKELSE VED OPPSTART PLS
LD P_On
TIM 0905 #100  ; FORSINKET STARTSIGNAL 999.06  VED OPPSTART AV PLS
AND PLS_FORSINKET_START_T  ; FORSINKET STARTSIGNAL 999.06  VED OPPSTART AV PLS
OUT PLS_INNFORSINK  ; FORSINKET SIGNAL VED OPPSTART AV pls
; rung 1: BLINK=1
LD P_On
OUT TR0
ANDNOT BLIK_TID2_S
TIM 0871 #5  ; BLIK_TID1_S
LD TR0
ANDNOT BLIK_TID1_S
OUT BLINK  ; 0,5 SEKUNERS BINK
; rung 2: HURTIGBLINKBLINK=1
LD P_On
OUT TR0
ANDNOT BLINK_HURTIG  ; 0.2S BLINK
TIM 0895 #2  ; 0.2S BLINK
LD TR0
ANDNOT BLINK_HURTIG  ; 0.2S BLINK
OUT HURTIG_BLINK  ; 0,2 SEKUNERS BINK
; rung 3: BLINRESET
LD BLIK_TID1_S
TIM 0872 #5  ; BLIK_TID2_S

### Section SUM_LINJEFEIL_NODE_4

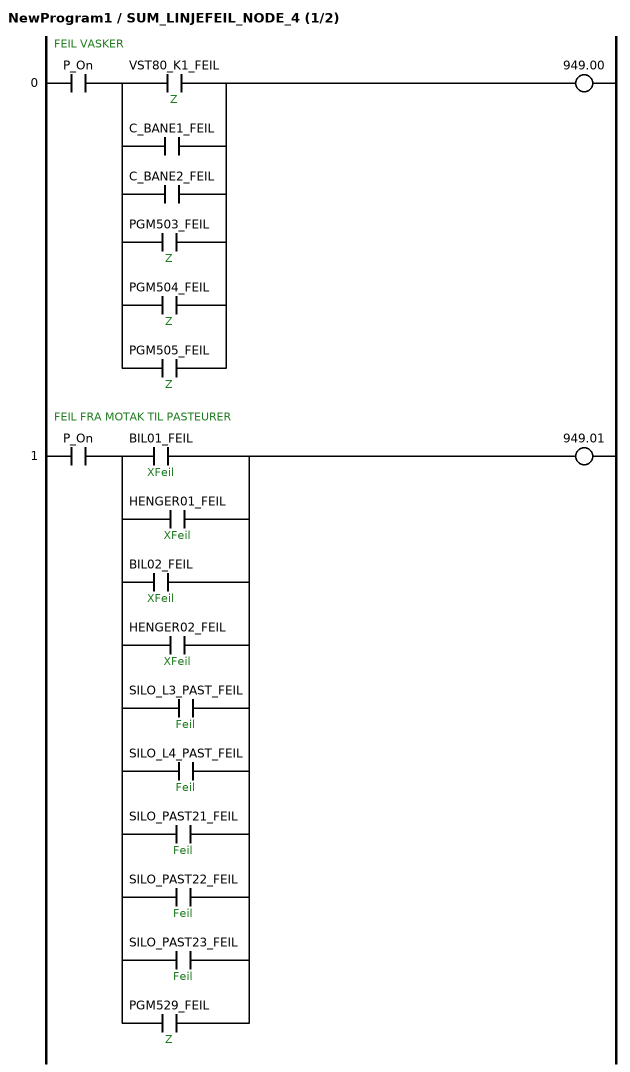
; rung 0: FEIL VASKER
LD P_On
LD VST80_K1_FEIL  ; Z
OR C_BANE1_FEIL
OR C_BANE2_FEIL
OR PGM503_FEIL  ; Z
OR PGM504_FEIL  ; Z
OR PGM505_FEIL  ; Z
ANDLD
OUT 949.00
; rung 1: FEIL FRA MOTAK TIL PASTEURER
LD P_On
LD BIL01_FEIL  ; XFeil
OR HENGER01_FEIL  ; XFeil
OR BIL02_FEIL  ; XFeil
OR HENGER02_FEIL  ; XFeil
OR SILO_L3_PAST_FEIL  ; Feil
OR SILO_L4_PAST_FEIL  ; Feil
OR SILO_PAST21_FEIL  ; Feil
OR SILO_PAST22_FEIL  ; Feil
OR SILO_PAST23_FEIL  ; Feil
OR PGM529_FEIL  ; Z
ANDLD
OUT 949.01

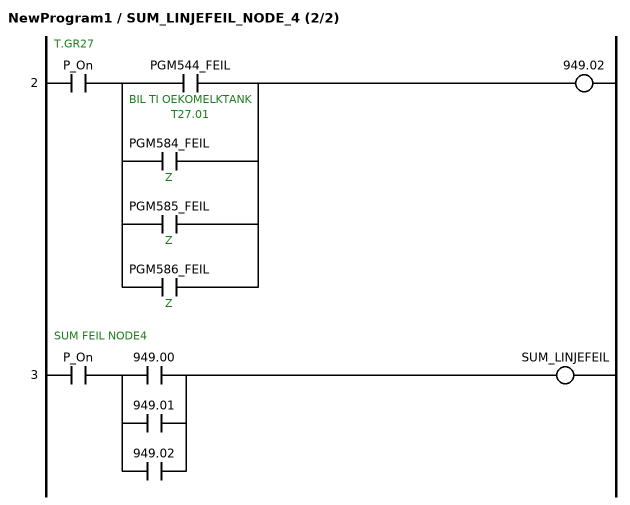
; rung 2: T.GR27
LD P_On
LD PGM544_FEIL  ; BIL TI OEKOMELKTANK T27.01
OR PGM584_FEIL  ; Z
OR PGM585_FEIL  ; Z
OR PGM586_FEIL  ; Z
ANDLD
OUT 949.02
; rung 3: SUM FEIL NODE4
LD P_On
LD 949.00
OR 949.01
OR 949.02
ANDLD
OUT SUM_LINJEFEIL

### Section VST80_LUT_DESINFEKT_FORBRUK

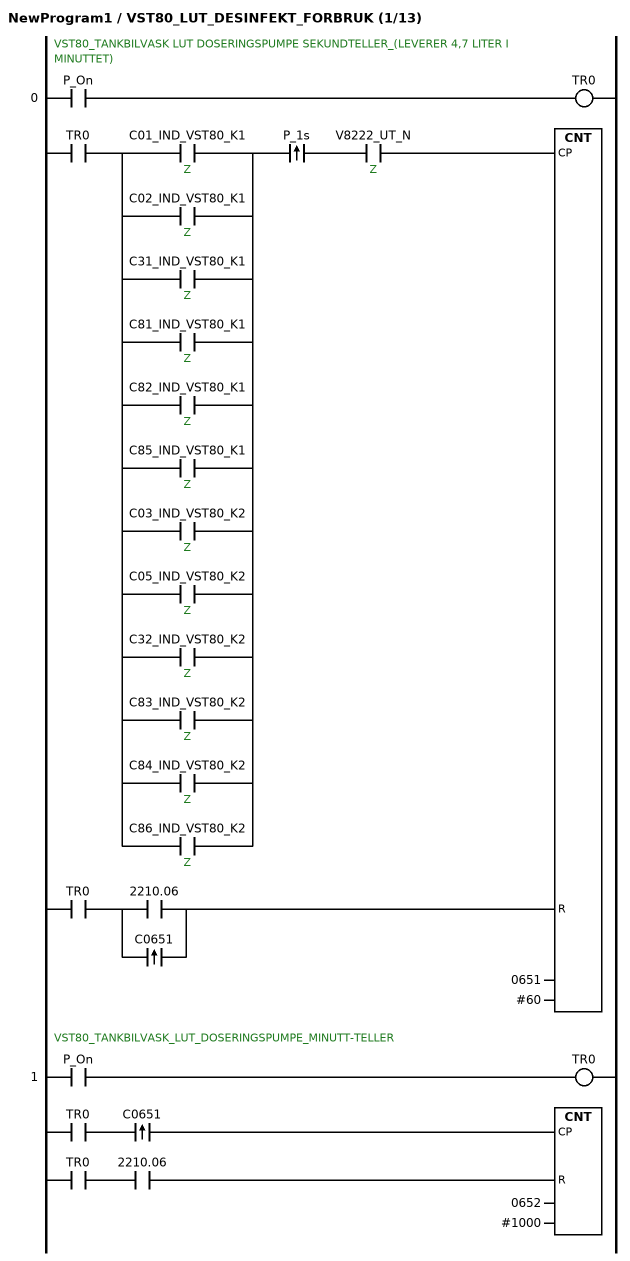
; rung 0: VST80_TANKBILVASK LUT DOSERINGSPUMPE SEKUNDTELLER_(LEVERER 4,7 LITER I MINUTTET)
LD P_On
OUT TR0
LD C01_IND_VST80_K1  ; Z
OR C02_IND_VST80_K1  ; Z
OR C31_IND_VST80_K1  ; Z
OR C81_IND_VST80_K1  ; Z
OR C82_IND_VST80_K1  ; Z
OR C85_IND_VST80_K1  ; Z
OR C03_IND_VST80_K2  ; Z
OR C05_IND_VST80_K2  ; Z
OR C32_IND_VST80_K2  ; Z
OR C83_IND_VST80_K2  ; Z
OR C84_IND_VST80_K2  ; Z
OR C86_IND_VST80_K2  ; Z
ANDLD
@AND P_1s
AND V8222_UT_N  ; Z
LD TR0
LD 2210.06
@OR C0651
ANDLD
CNT 0651 #60
; rung 1: VST80_TANKBILVASK_LUT_DOSERINGSPUMPE_MINUTT-TELLER
LD P_On
OUT TR0
@AND C0651
LD TR0
AND 2210.06
CNT 0652 #1000

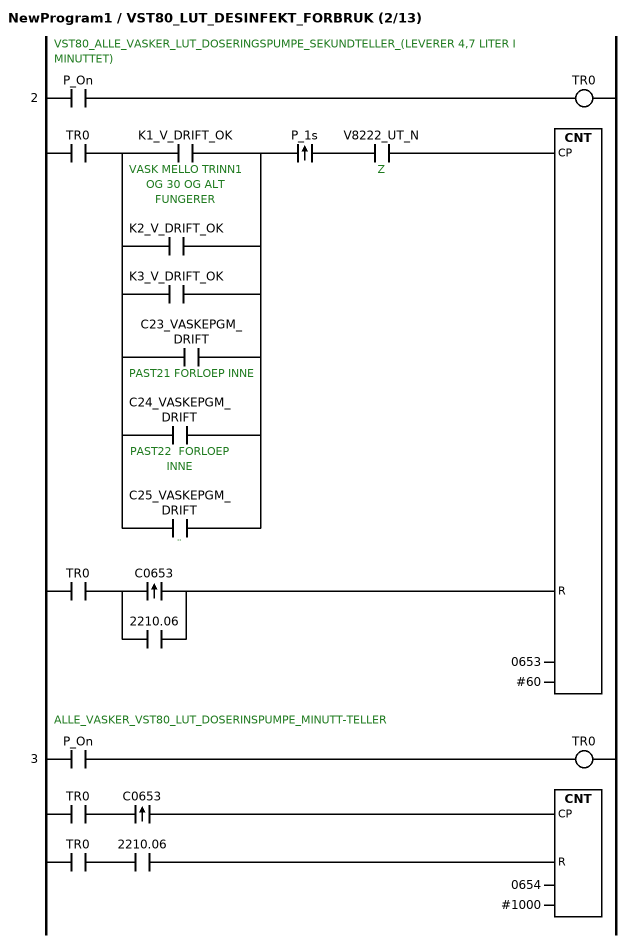
; rung 2: VST80_ALLE_VASKER_LUT_DOSERINGSPUMPE_SEKUNDTELLER_(LEVERER 4,7 LITER I MINUTTET)
LD P_On
OUT TR0
LD K1_V_DRIFT_OK  ; VASK MELLO TRINN1 OG 30 OG ALT FUNGERER
OR K2_V_DRIFT_OK
OR K3_V_DRIFT_OK
OR C23_VASKEPGM_DRIFT  ; PAST21 FORLOEP INNE
OR C24_VASKEPGM_DRIFT  ; PAST22  FORLOEP INNE
OR C25_VASKEPGM_DRIFT  ; ¨
ANDLD
@AND P_1s
AND V8222_UT_N  ; Z
LD TR0
@LD C0653
OR 2210.06
ANDLD
CNT 0653 #60
; rung 3: ALLE_VASKER_VST80_LUT_DOSERINSPUMPE_MINUTT-TELLER
LD P_On
OUT TR0
@AND C0653
LD TR0
AND 2210.06
CNT 0654 #1000

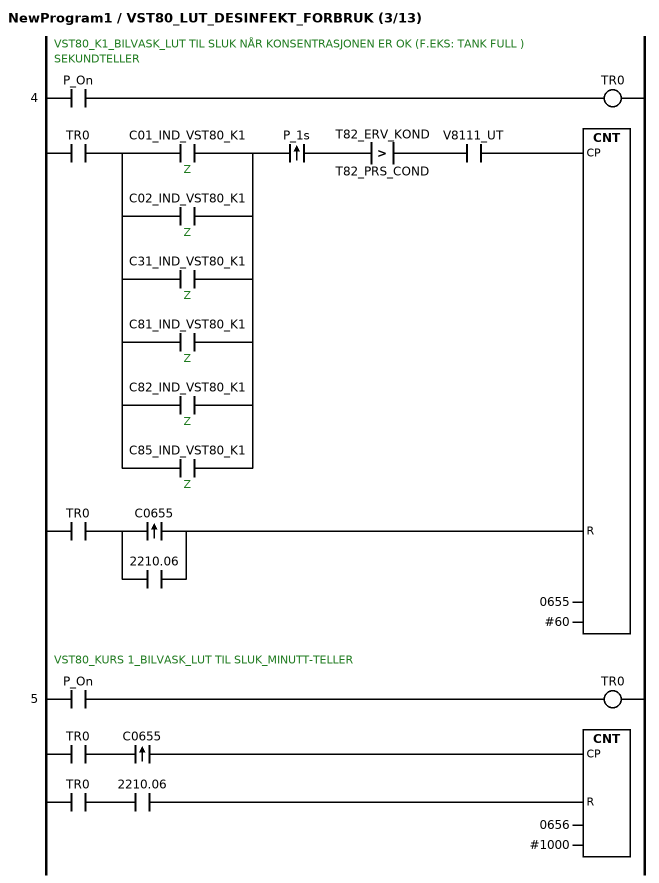
; rung 4: VST80_K1_BILVASK_LUT TIL SLUK NÅR KONSENTRASJONEN ER OK (F.EKS: TANK FULL ) SEKUNDTELLER
LD P_On
OUT TR0
LD C01_IND_VST80_K1  ; Z
OR C02_IND_VST80_K1  ; Z
OR C31_IND_VST80_K1  ; Z
OR C81_IND_VST80_K1  ; Z
OR C82_IND_VST80_K1  ; Z
OR C85_IND_VST80_K1  ; Z
ANDLD
@AND P_1s
AND>(320) T82_ERV_KOND T82_PRS_COND
AND V8111_UT
LD TR0
@LD C0655
OR 2210.06
ANDLD
CNT 0655 #60
; rung 5: VST80_KURS 1_BILVASK_LUT TIL SLUK_MINUTT-TELLER
LD P_On
OUT TR0
@AND C0655
LD TR0
AND 2210.06
CNT 0656 #1000

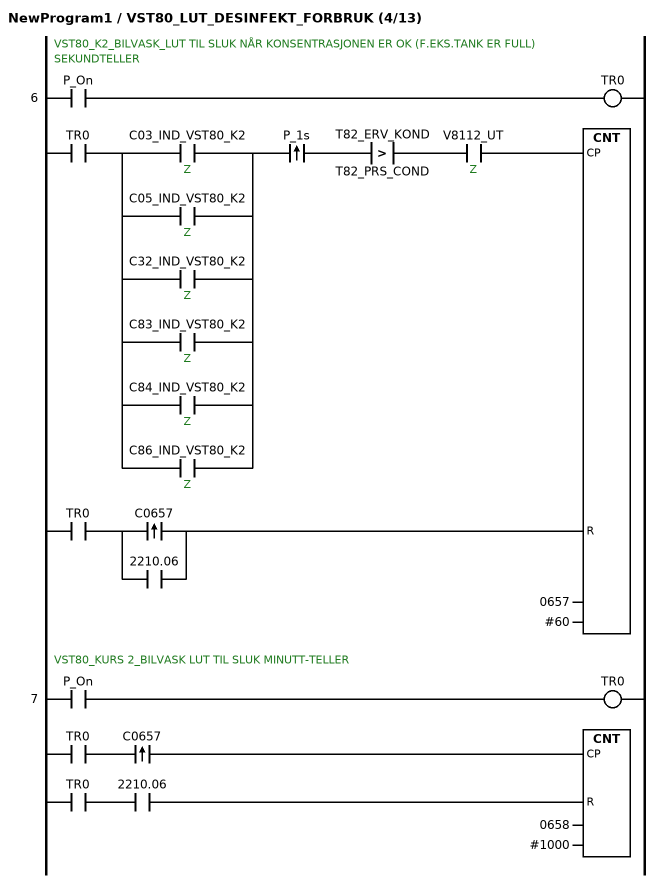
; rung 6: VST80_K2_BILVASK_LUT TIL SLUK NÅR KONSENTRASJONEN ER OK (F.EKS.TANK ER FULL) SEKUNDTELLER
LD P_On
OUT TR0
LD C03_IND_VST80_K2  ; Z
OR C05_IND_VST80_K2  ; Z
OR C32_IND_VST80_K2  ; Z
OR C83_IND_VST80_K2  ; Z
OR C84_IND_VST80_K2  ; Z
OR C86_IND_VST80_K2  ; Z
ANDLD
@AND P_1s
AND>(320) T82_ERV_KOND T82_PRS_COND
AND V8112_UT  ; Z
LD TR0
@LD C0657
OR 2210.06
ANDLD
CNT 0657 #60
; rung 7: VST80_KURS 2_BILVASK LUT TIL SLUK MINUTT-TELLER
LD P_On
OUT TR0
@AND C0657
LD TR0
AND 2210.06
CNT 0658 #1000

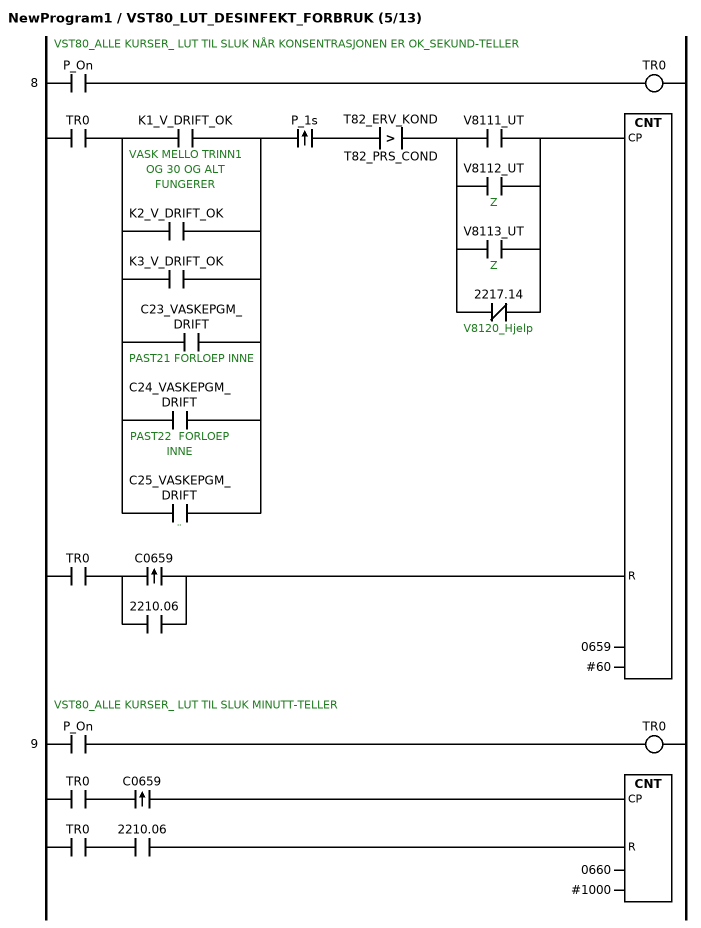
; rung 8: VST80_ALLE KURSER_ LUT TIL SLUK NÅR KONSENTRASJONEN ER OK_SEKUND-TELLER
LD P_On
OUT TR0
LD K1_V_DRIFT_OK  ; VASK MELLO TRINN1 OG 30 OG ALT FUNGERER
OR K2_V_DRIFT_OK
OR K3_V_DRIFT_OK
OR C23_VASKEPGM_DRIFT  ; PAST21 FORLOEP INNE
OR C24_VASKEPGM_DRIFT  ; PAST22  FORLOEP INNE
OR C25_VASKEPGM_DRIFT  ; ¨
ANDLD
@AND P_1s
AND>(320) T82_ERV_KOND T82_PRS_COND
LD V8111_UT
OR V8112_UT  ; Z
OR V8113_UT  ; Z
ORNOT 2217.14  ; V8120_Hjelp
ANDLD
LD TR0
@LD C0659
OR 2210.06
ANDLD
CNT 0659 #60
; rung 9: VST80_ALLE KURSER_ LUT TIL SLUK MINUTT-TELLER
LD P_On
OUT TR0
@AND C0659
LD TR0
AND 2210.06
CNT 0660 #1000

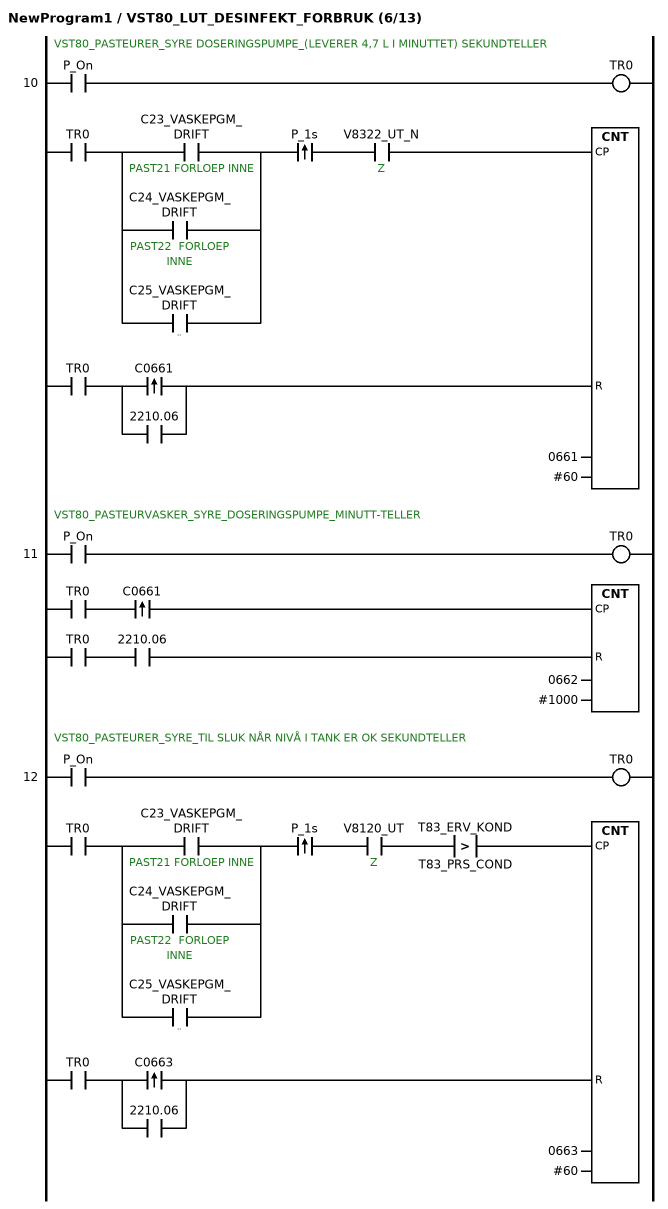
; rung 10: VST80_PASTEURER_SYRE DOSERINGSPUMPE_(LEVERER 4,7 L I MINUTTET) SEKUNDTELLER
LD P_On
OUT TR0
LD C23_VASKEPGM_DRIFT  ; PAST21 FORLOEP INNE
OR C24_VASKEPGM_DRIFT  ; PAST22  FORLOEP INNE
OR C25_VASKEPGM_DRIFT  ; ¨
ANDLD
@AND P_1s
AND V8322_UT_N  ; Z
LD TR0
@LD C0661
OR 2210.06
ANDLD
CNT 0661 #60
; rung 11: VST80_PASTEURVASKER_SYRE_DOSERINGSPUMPE_MINUTT-TELLER
LD P_On
OUT TR0
@AND C0661
LD TR0
AND 2210.06
CNT 0662 #1000
; rung 12: VST80_PASTEURER_SYRE_TIL SLUK NÅR NIVÅ I TANK ER OK SEKUNDTELLER
LD P_On
OUT TR0
LD C23_VASKEPGM_DRIFT  ; PAST21 FORLOEP INNE
OR C24_VASKEPGM_DRIFT  ; PAST22  FORLOEP INNE
OR C25_VASKEPGM_DRIFT  ; ¨
ANDLD
@AND P_1s
AND V8120_UT  ; Z
AND>(320) T83_ERV_KOND T83_PRS_COND
LD TR0
@LD C0663
OR 2210.06
ANDLD
CNT 0663 #60

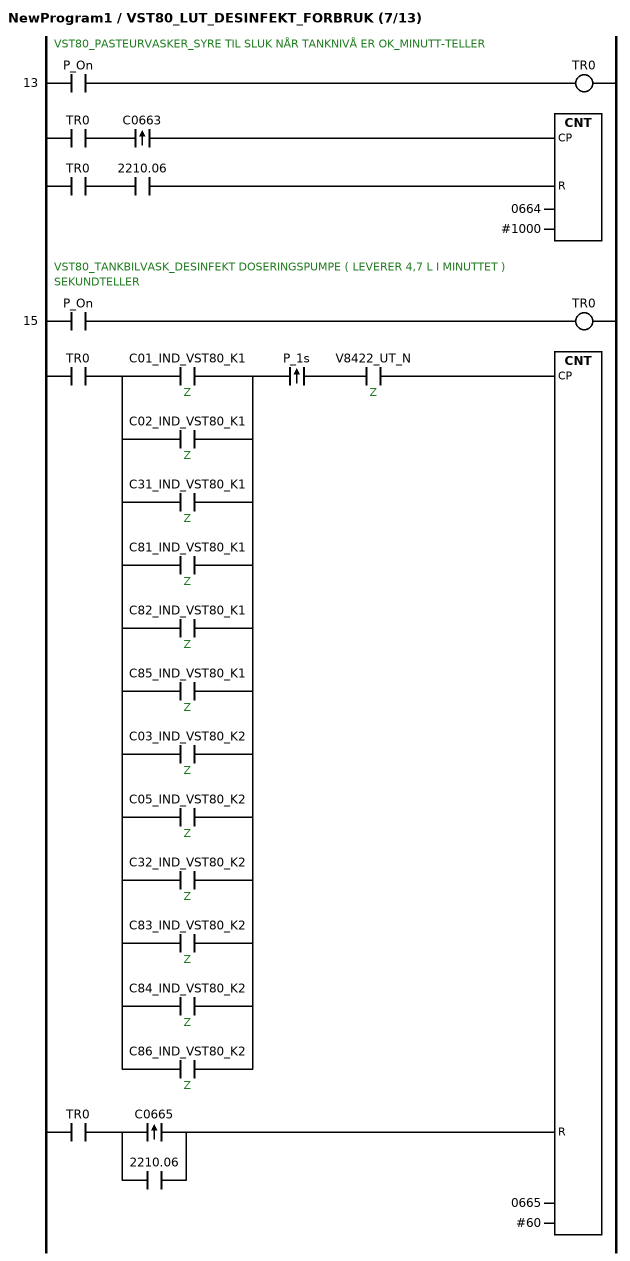
; rung 13: VST80_PASTEURVASKER_SYRE TIL SLUK NÅR TANKNIVÅ ER OK_MINUTT-TELLER
LD P_On
OUT TR0
@AND C0663
LD TR0
AND 2210.06
CNT 0664 #1000
; rung 14
; rung 15: VST80_TANKBILVASK_DESINFEKT DOSERINGSPUMPE ( LEVERER 4,7 L I MINUTTET ) SEKUNDTELLER
LD P_On
OUT TR0
LD C01_IND_VST80_K1  ; Z
OR C02_IND_VST80_K1  ; Z
OR C31_IND_VST80_K1  ; Z
OR C81_IND_VST80_K1  ; Z
OR C82_IND_VST80_K1  ; Z
OR C85_IND_VST80_K1  ; Z
OR C03_IND_VST80_K2  ; Z
OR C05_IND_VST80_K2  ; Z
OR C32_IND_VST80_K2  ; Z
OR C83_IND_VST80_K2  ; Z
OR C84_IND_VST80_K2  ; Z
OR C86_IND_VST80_K2  ; Z
ANDLD
@AND P_1s
AND V8422_UT_N  ; Z
LD TR0
@LD C0665
OR 2210.06
ANDLD
CNT 0665 #60

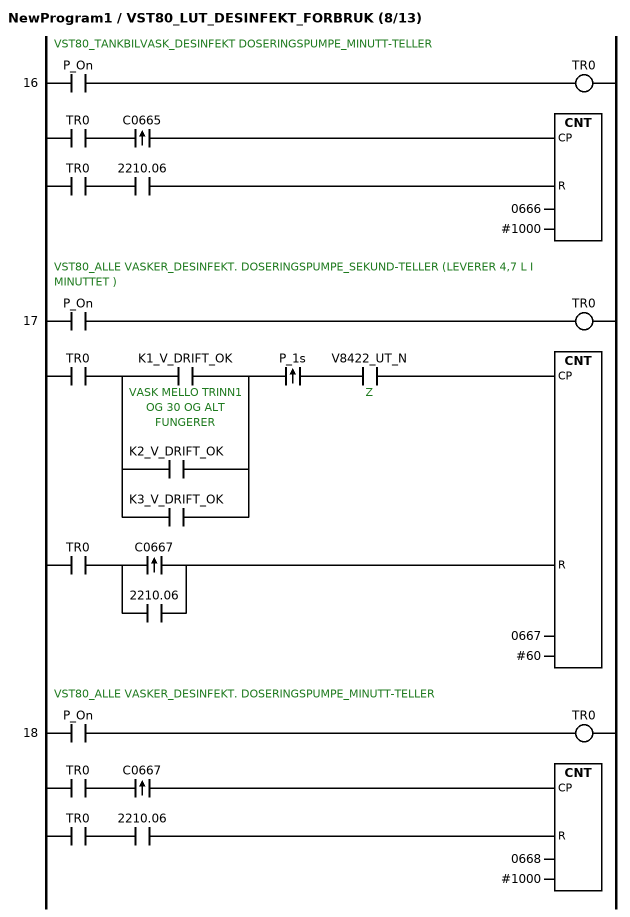
; rung 16: VST80_TANKBILVASK_DESINFEKT DOSERINGSPUMPE_MINUTT-TELLER
LD P_On
OUT TR0
@AND C0665
LD TR0
AND 2210.06
CNT 0666 #1000
; rung 17: VST80_ALLE VASKER_DESINFEKT. DOSERINGSPUMPE_SEKUND-TELLER (LEVERER 4,7 L I MINUTTET )
LD P_On
OUT TR0
LD K1_V_DRIFT_OK  ; VASK MELLO TRINN1 OG 30 OG ALT FUNGERER
OR K2_V_DRIFT_OK
OR K3_V_DRIFT_OK
ANDLD
@AND P_1s
AND V8422_UT_N  ; Z
LD TR0
@LD C0667
OR 2210.06
ANDLD
CNT 0667 #60
; rung 18: VST80_ALLE VASKER_DESINFEKT. DOSERINGSPUMPE_MINUTT-TELLER
LD P_On
OUT TR0
@AND C0667
LD TR0
AND 2210.06
CNT 0668 #1000

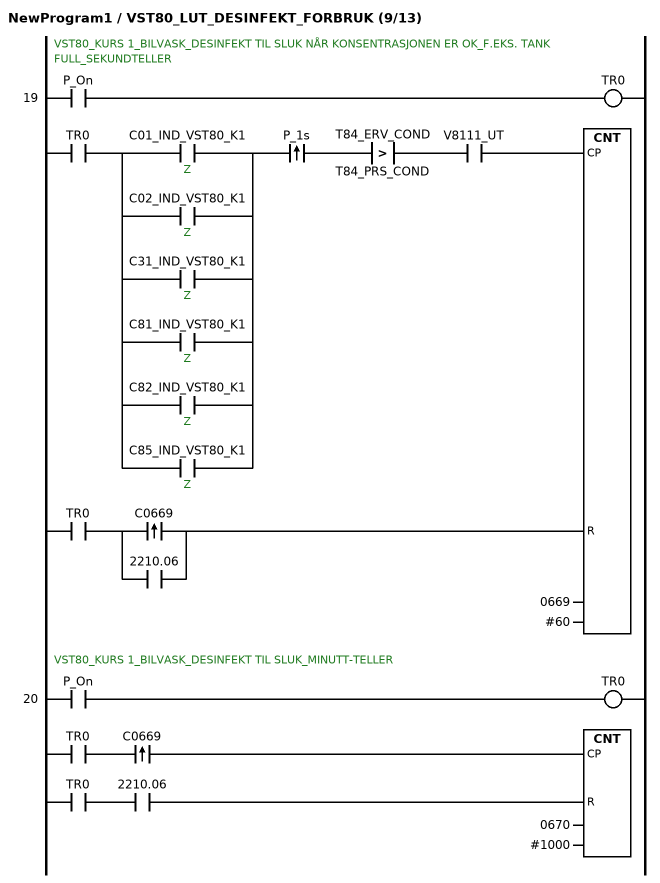
; rung 19: VST80_KURS 1_BILVASK_DESINFEKT TIL SLUK NÅR KONSENTRASJONEN ER OK_F.EKS. TANK FULL_SEKUNDTELLER
LD P_On
OUT TR0
LD C01_IND_VST80_K1  ; Z
OR C02_IND_VST80_K1  ; Z
OR C31_IND_VST80_K1  ; Z
OR C81_IND_VST80_K1  ; Z
OR C82_IND_VST80_K1  ; Z
OR C85_IND_VST80_K1  ; Z
ANDLD
@AND P_1s
AND>(320) T84_ERV_COND T84_PRS_COND
AND V8111_UT
LD TR0
@LD C0669
OR 2210.06
ANDLD
CNT 0669 #60
; rung 20: VST80_KURS 1_BILVASK_DESINFEKT TIL SLUK_MINUTT-TELLER
LD P_On
OUT TR0
@AND C0669
LD TR0
AND 2210.06
CNT 0670 #1000

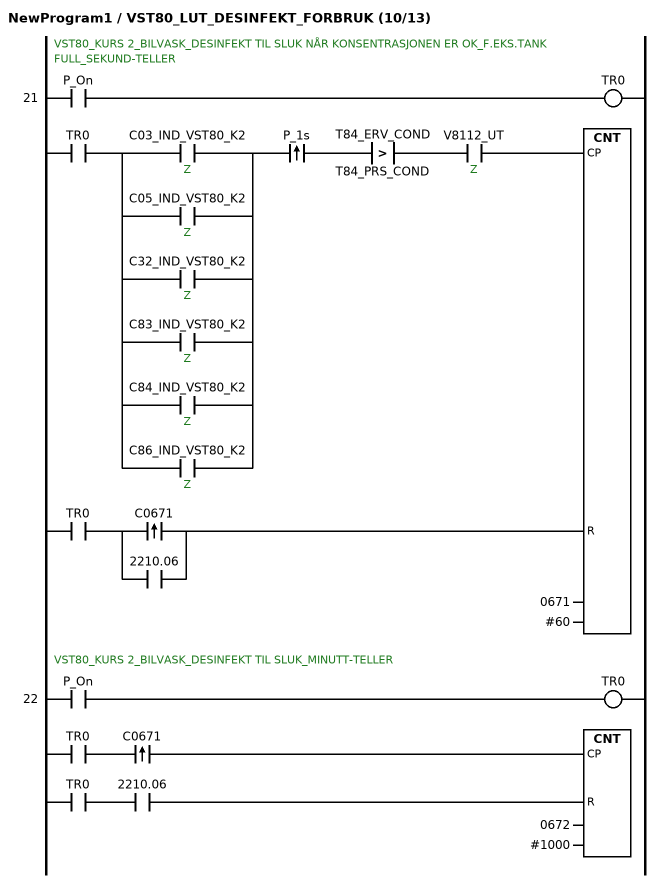
; rung 21: VST80_KURS 2_BILVASK_DESINFEKT TIL SLUK NÅR KONSENTRASJONEN ER OK_F.EKS.TANK FULL_SEKUND-TELLER
LD P_On
OUT TR0
LD C03_IND_VST80_K2  ; Z
OR C05_IND_VST80_K2  ; Z
OR C32_IND_VST80_K2  ; Z
OR C83_IND_VST80_K2  ; Z
OR C84_IND_VST80_K2  ; Z
OR C86_IND_VST80_K2  ; Z
ANDLD
@AND P_1s
AND>(320) T84_ERV_COND T84_PRS_COND
AND V8112_UT  ; Z
LD TR0
@LD C0671
OR 2210.06
ANDLD
CNT 0671 #60
; rung 22: VST80_KURS 2_BILVASK_DESINFEKT TIL SLUK_MINUTT-TELLER
LD P_On
OUT TR0
@AND C0671
LD TR0
AND 2210.06
CNT 0672 #1000

